FUNCTION_BLOCK EL3142
VAR
	_io : EL3xx2_Data;
	{attribute addProperty Name "WcState"}
	_wcState : WcStateInputToggle;
	{attribute addProperty Name "Info data"}
	_infoData : InfoDataAds;
END_VAR

PROPERTY IO : REFERENCE TO EL3xx2_Data
GET
IO REF= _io;
END_GET
END_PROPERTY

PROPERTY WcState : REFERENCE TO WcStateInputToggle
GET
WcState REF= _wcState;
END_GET
END_PROPERTY

END_FUNCTION_BLOCK

(* stored: Version 1.1.0.1, ProductVersion 3.1.4024.9
   POU EL3142: Id {63c9e7d0-4f06-0410-2dcb-3a583ddf2794}, SpecialFunc None
   Property IO: Id {3e07552d-a6a7-0433-2a0d-0bdcac826b7a}
   Get Get: Id {cbb68fe0-0f22-0cd1-0f27-adaeb8e2704a}
   Property WcState: Id {8783a5c1-e66f-0b7f-15ee-d598e0ebd4de}
   Get Get: Id {d6ed5d5e-fbae-0fdd-2b34-cf12f95bb0c5} *)
